FUNCTION_BLOCK Service
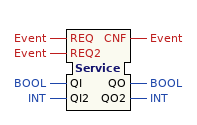
  EVENT_INPUT
    REQ;
    REQ2;
  END_EVENT
  EVENT_OUTPUT
    CNF;
  END_EVENT
  VAR_INPUT
    QI : BOOL;
    QI2 : INT;
  END_VAR
  VAR_OUTPUT
    QO : BOOL;
    QO2 : INT;
  END_VAR
END_FUNCTION_BLOCK
